PROGRAM MAIN
VAR
END_VAR

Alias();
AnalogConversion();
Sequence();

END_PROGRAM

(* stored: Version 1.1.0.1, ProductVersion 3.1.4024.11
   POU MAIN: Id {b3538f2d-ba7d-49bb-a337-3cef62914be8}, SpecialFunc None *)
